TYPE ST_StorageSlot :
STRUCT
	nStorageId : INT;
	nStorageName : STRING;
	bMaintanence : BOOL;
END_STRUCT
END_TYPE

(* stored: Version 1.1.0.1, ProductVersion 3.1.4024.16
   DUT ST_StorageSlot: Id {b5dd1852-5236-4d8f-a0bb-da0d258b9e17} *)
